//PLC 2
PROGRAM MAIN
VAR
END_VAR

F_ConsumeTime(400);

END_PROGRAM

(* stored: Version 1.1.0.1, ProductVersion 3.1.4026.18
   POU MAIN: Id {c6961578-a6b4-4672-aad6-a12fe19225da}, SpecialFunc None *)
